FUNCTION_BLOCK EV_Scale (* Typed view of Scale's state channel (inputs and holder) *)
  (* Standard: 61499-2 *)
  (* Version 0.1, 2026-09-28, Project contributors, AAU Smart Production Lab *)
  PACKAGE filling;
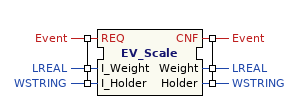
  EVENT_INPUT
    REQ WITH I_Weight, I_Holder;
  END_EVENT
  EVENT_OUTPUT
    CNF WITH Weight, Holder;
  END_EVENT
  VAR_INPUT
    I_Weight : LREAL;
    I_Holder : WSTRING;
  END_VAR
  VAR_OUTPUT
    Weight : LREAL;
    Holder : WSTRING;
  END_VAR
  EC_STATES
    REQ : REQ -> CNF;
  END_STATES
  ALGORITHM REQ IN ST:
Weight := I_Weight;
Holder := I_Holder;
  END_ALGORITHM
END_FUNCTION_BLOCK
